(* CoDeSys 2.3 export: POSE6.EXP *)

(* Data type in MNG_TCPIP *)
TYPE POSE6 :(* position and orientation as an euler based pose *)
STRUCT
	x, y, z, a, b, c : REAL;
END_STRUCT
END_TYPE
